PROGRAM P3_01_BatchData
VAR
END_VAR
VAR PERSISTENT
	dtBatchOpen					:DT;
	dtBatchClose				:DT;
	
	ulBatchOpen					:ULINT;
	ulBatchClose				:ULINT;
END_VAR
VAR // added by the converter: edge detectors and wires of the graphical bodies
    _rt1, _rt2 : R_TRIG;
    _w1, _w2 : BOOL;
END_VAR

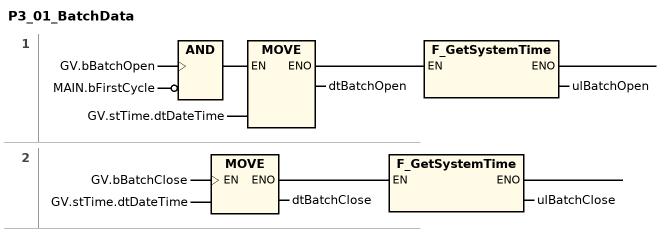
// NETWORK 1
_rt1(CLK := GV.bBatchOpen);
_w1 := _rt1.Q AND NOT MAIN.bFirstCycle;
IF _w1 THEN dtBatchOpen := GV.stTime.dtDateTime; END_IF
IF _w1 THEN ulBatchOpen := F_GetSystemTime(); END_IF

// NETWORK 2
_rt2(CLK := GV.bBatchClose);
_w2 := _rt2.Q;
IF _w2 THEN dtBatchClose := GV.stTime.dtDateTime; END_IF
IF _w2 THEN ulBatchClose := F_GetSystemTime(); END_IF

END_PROGRAM

(* stored: Version 1.1.0.1, ProductVersion 3.1.4024.12
   POU P3_01_BatchData: Id {4e51726e-df01-47a9-941f-6342ec7bf293}, SpecialFunc None *)
